PROGRAM PRG_3
VAR
	nCount: INT ;
	nCount2: INT ;
	fbprg : FB_PRG;
	
END_VAR
VAR
	
END_VAR

nCount := nCOunt +1;

 fbprg();

END_PROGRAM

(* stored: Version 1.1.0.1, ProductVersion 3.1.4024.16
   POU PRG_3: Id {e59885e0-22a5-4b72-81b0-3ca279aa34e3}, SpecialFunc None *)
